# EPICS autosave request: DG645/iocBoot/iocDG645-IOC-01/dgconfigMenu.req
file configMenu.req P=$(P),CONFIG=$(CONFIG)
file dgconfig_settings.req
